TYPE TRunCmdSharpen :
	(
		RCS_None,
		RCS_MoveStep
	);
END_TYPE

(* stored: Version 1.1.0.1, ProductVersion 3.1.4022.12
   DUT TRunCmdSharpen: Id {c2c34ebc-86b2-401e-a9bb-2b05fb3c0de7} *)
